{attribute 'qualified_only'}
VAR_GLOBAL CONSTANT
	OBSERVER_CNT:	INT := 5;
END_VAR

(* stored: Version 1.1.0.1, ProductVersion 3.1.4026.18
   GVL GVL_GENERIC_OBSERVER: Id {1642046f-7beb-4651-a666-192ef7393ff6} *)
